# EPICS autosave request: iocBoot/gmca_23i_ioc1/dbSave/robot.req
% $(P)pause
$(P)gh_pos
$(P)gy_pos
$(P)tmoh
$(P)tmoc
$(P)senh
$(P)senc
